// Implicitly generated code : DO NOT EDIT
FUNCTION CheckRangeUnsigned : UDINT
VAR_INPUT
	value, lower, upper: UDINT;
END_VAR
VAR
    sMessageLow   : STRING := 'CheckRangeUnsigned: Value too low (%d)';
    sMessageHigh  : STRING := 'CheckRangeUnsigned: Value too high (%d)';
END_VAR

// Implicitly generated code : Only an Implementation suggestion
{noflow}
IF (value < lower) THEN
	CheckRangeUnsigned := lower;
	// Log message
	ADSLOGDINT(msgCtrlMask := ADSLOG_MSGTYPE_WARN,
               msgFmtStr   := sMessageLow,
               dintArg     := TO_INT(value));
ELSIF(value > upper) THEN
	CheckRangeUnsigned := upper;
	// Log message
    ADSLOGDINT(msgCtrlMask := ADSLOG_MSGTYPE_WARN,
               msgFmtStr   := sMessageHigh,
               dintArg     := TO_INT(value));
ELSE
	CheckRangeUnsigned := value;
END_IF
{flow}

END_FUNCTION

(* stored: Version 1.1.0.1, ProductVersion 3.1.4024.11
   POU CheckRangeUnsigned: Id {ae40ae72-7d8f-4e7f-ac70-1a1fe2614d5d}, SpecialFunc CheckRangeUnsigned *)
